TYPE InfoDataAdsAddrStateBase_1916E49F :
STRUCT
END_STRUCT
END_TYPE
